(* CODESYS project Vision.library
   Version: 2025.10.24.3
   Description: Disable checks for trigger
   Title: Vision
   Placeholder: Vision
   Company: Photara

Project tree, tasks and I/O mapping:
  libraries: Base, * (Photara); Tc2_Standard, * (Beckhoff Automation GmbH); Tc2_System, * (Beckhoff Automation GmbH); TcUnit, * (www.tcunit.org)
  DUTs/
    data type ST_PyADSAPI
    data type ST_VisionConfiguration
    data type ST_VisionResults
    data type ST_VisionStatus
  GVLs/
    global variables GC_Vision
    global variables GPL_Vision
  ITFs/
    interface I_Vision: P_HandshakeStatus, P_VisionStatus, Reset, Trigger
    interface I_VisionConfiguration: P_VisionConfiguration
  POUs/
    function block FB_ADSVision [ST]: Busy, CyclicLogic, Error, Reset, P_HandshakeStatus, P_VisionConfiguration, P_VisionStatus, Trigger, _InitializeReferences, _EvaluateCompletionConditions, _FourBitHandshake, _SetCommandPermIntlkConfiguration, _Trigger, _UpdateComponentStatus, P_TP_PyAds
    program MAIN [ST]
    program PRG_TEST [ST]
  Tests/
    function block FB_VisionTests [ST]: TEST_GivenFullCycle_WhenTriggerToResultComplete_ExpectCorrectStateTransition, TEST_GivenIdle_WhenTriggerCalled_ExpectStartTriggerRaised, TEST_GivenInvalidData_WhenResultReady_ExpectErrorCodeBadData, TEST_GivenMultipleCycles_WhenSequentialRuns_ExpectNoStateLeak, TEST_GivenRapidTriggerResetSequence_ExpectNoRaceConditions, TEST_GivenResetCalled_WhenBusy_ExpectReturnToIdle, TEST_GivenResultReady_WhenResultNotConsumed_ExpectTimeoutFault, TEST_GivenResultReady_WhenResultsLatched_ExpectResultsReceivedRaised, TEST_GivenResultReady_WhenResultsValid_ExpectResultsLatched, TEST_GivenResults_WhenValid_ExpectBusyFalseAtHandshakeCompletion, TEST_GivenResultsReceived_WhenVisionClearsResultReady_ExpectAckCleared, TEST_GivenTrigger_WhenAckNeverComes_ExpectErrorCodeTimeout, TEST_GivenTriggerAckReceived_WhenTriggerActive_ExpectStartTriggerCleared, TEST_GivenTriggerCycleComplete_ExpectReturnToIdle, TEST_GivenTriggerSent_WhenAckNotReceived_ExpectTimeoutFault, TEST_GivenTriggerWhileBusy_ExpectRejected, TEST_GivenVisionClearsEarly_WhenResultsNotConsumed_ExpectSafeIdle
*)

// DUTs/ST_PyADSAPI
TYPE ST_PyADSAPI :
STRUCT
	StartTrigger		: BOOL;
	TriggerAck			: BOOL;
	ResultsReady		: BOOL;
	ResultsReceived		: BOOL;
	
	VisionResult        : ST_VisionResults;
END_STRUCT
END_TYPE

// DUTs/ST_VisionConfiguration
TYPE ST_VisionConfiguration :
STRUCT
	ComponentConfiguration : REFERENCE TO ST_ComponentConfiguration;
END_STRUCT
END_TYPE

// DUTs/ST_VisionResults
TYPE ST_VisionResults :
STRUCT
	TargetX			: REAL;
    TargetY			: REAL;
    TargetTheta		: REAL;
	
	ResultCode      : BYTE;
END_STRUCT
END_TYPE

// DUTs/ST_VisionStatus
TYPE ST_VisionStatus :
STRUCT
	ComponentStatus 	: REFERENCE TO ST_ComponentStatus;
	VisionResult		: ST_VisionResults;
	
END_STRUCT
END_TYPE

// GVLs/GC_Vision
{attribute 'qualified_only'}
{attribute 'global_init_slot' := '40620'}
VAR_GLOBAL CONSTANT
	INDEX_COMMAND_MIN				: DINT := GPL_Vision.INDEX_COMMAND_MIN;
	INDEX_COMMAND_MAX				: DINT := GPL_Vision.INDEX_COMMAND_MAX;
END_VAR

// GVLs/GPL_Vision
{attribute 'qualified_only'}
{attribute 'global_init_slot' := '40520'}
VAR_GLOBAL CONSTANT
	INDEX_COMMAND_MIN				: DINT := 0;
	INDEX_COMMAND_MAX				: DINT := 1;
END_VAR

// ITFs/I_Vision
INTERFACE I_Vision EXTENDS Base.I_BaseCyclic

PROPERTY P_HandshakeStatus : REFERENCE TO ST_PyADSAPI
GET
END_GET
END_PROPERTY

PROPERTY P_VisionStatus : REFERENCE TO ST_VisionStatus
GET
END_GET
END_PROPERTY

METHOD Reset: Base.E_CommandResult
VAR_INPUT
END_VAR
END_METHOD

METHOD Trigger : BOOL
VAR_INPUT
END_VAR
END_METHOD

END_INTERFACE

// ITFs/I_VisionConfiguration
INTERFACE I_VisionConfiguration EXTENDS __SYSTEM.IQueryInterface

PROPERTY P_VisionConfiguration : REFERENCE TO ST_VisionConfiguration
GET
END_GET
END_PROPERTY

END_INTERFACE

// POUs/FB_ADSVision
{attribute 'no_explicit_call' := 'do not call this POU directly'} 
FUNCTION_BLOCK FB_ADSVision EXTENDS FB_Component<GC_Vision.INDEX_COMMAND_MIN, GC_Vision.INDEX_COMMAND_MAX> IMPLEMENTS I_Vision, I_VisionConfiguration
VAR CONSTANT
	INDEX_CMD_TRIGGER		: DINT := 0;
END_VAR
VAR
	VisionConfiguration 	: ST_VisionConfiguration;
	VisionStatus 			: ST_VisionStatus;
	PyVars 					: ST_PyADSAPI;
END_VAR

PROPERTY Busy : BOOL
GET
// Combine base busy state (command execution) with handshake flags
Busy := SUPER^.Busy OR PyVars.StartTrigger OR PyVars.TriggerAck OR PyVars.ResultsReady OR PyVars.ResultsReceived;
END_GET
END_PROPERTY

METHOD CyclicLogic
SUPER^.CyclicLogic();

_UpdateComponentStatus();
END_METHOD

PROPERTY Error : BOOL
GET
IF SUPER^.iCommands[INDEX_CMD_TRIGGER] <> 0 THEN
	Error := SUPER^.iCommands[INDEX_CMD_TRIGGER].P_CommandStatus.Result = Base.E_CommandResult.RequestTimeout;
END_IF;
END_GET
END_PROPERTY

METHOD Reset : Base.E_CommandResult
// Clear all handshake flags first
PyVars.StartTrigger		:= FALSE;
PyVars.ResultsReceived	:= FALSE;
PyVars.TriggerAck		:= FALSE;
PyVars.ResultsReady		:= FALSE;

// Clear result values
PyVars.VisionResult.TargetTheta	:= 0;
PyVars.VisionResult.TargetX		:= 0;
PyVars.VisionResult.TargetY		:= 0;
PyVars.VisionResult.ResultCode    := 255; // 0xFF = uninitialized/reset state

// Force complete any busy command before reset
IF ComponentStatus.iLastCommand <> 0 THEN
    IF ComponentStatus.iLastCommand.Busy THEN
        ComponentStatus.iLastCommand.Abort();
    END_IF
END_IF

// Call base reset to clear command state
// Reset := SUPER^.Reset();
Reset := E_CommandResult.Ok;
END_METHOD

PROPERTY P_HandshakeStatus : REFERENCE TO ST_PyADSAPI
GET
P_HandshakeStatus	REF= PyVars;
END_GET
END_PROPERTY

PROPERTY P_VisionConfiguration : REFERENCE TO ST_VisionConfiguration
GET
P_VisionConfiguration	REF= VisionConfiguration;
END_GET
END_PROPERTY

PROPERTY P_VisionStatus : REFERENCE TO ST_VisionStatus
GET
P_VisionStatus REF= VisionStatus;
END_GET
END_PROPERTY

METHOD Trigger : BOOL
// ExecuteCommand(CmdIndex := INDEX_CMD_TRIGGER);
// 
// IF SUPER^.iCommands[INDEX_CMD_TRIGGER].P_CommandStatus.Result = Base.E_CommandResult.Accepted THEN
	Trigger	:= _Trigger();
// END_IF
END_METHOD

METHOD PROTECTED _InitializeReferences : BOOL
//Initialize data references
//Order is important!
BaseConfiguration.InstancePath 						REF= InstancePath;

ComponentConfiguration.BaseConfiguration 			REF= SUPER^.BaseConfiguration;
                                                    
ComponentStatus.BaseStatus							REF= SUPER^.BaseStatus;

ComponentStatus.AmsNetId							REF= ComponentConfiguration.AmsNetId;

VisionConfiguration.ComponentConfiguration			REF= SUPER^.ComponentConfiguration;

VisionStatus.ComponentStatus						REF= SUPER^.ComponentStatus;

_InitializeReferences 								:= TRUE; // apply at end of all reference initialization
END_METHOD

(*
Example Implementation:
// Set completion conditions - commands complete immediately after transitioning to acting state
// This prevents the component from staying busy and blocking other commands
SUPER^.CommandCompletionConditions[INDEX_COMMAND_ABORT]            		:= (SequencerStatus.CurrentState = E_PackMLState.Aborting);
SUPER^.CommandCompletionConditions[INDEX_COMMAND_CLEAR]            		:= (SequencerStatus.CurrentState = E_PackMLState.Clearing);
SUPER^.CommandCompletionConditions[INDEX_COMMAND_COMPLETE]         		:= (SequencerStatus.CurrentState = E_PackMLState.Completing);
SUPER^.CommandCompletionConditions[INDEX_COMMAND_HOLD]             		:= (SequencerStatus.CurrentState = E_PackMLState.Holding);
SUPER^.CommandCompletionConditions[INDEX_COMMAND_RESET]            		:= (SequencerStatus.CurrentState = E_PackMLState.Resetting);
SUPER^.CommandCompletionConditions[INDEX_COMMAND_RESUMEFROMHOLD]   		:= (SequencerStatus.CurrentState = E_PackMLState.Unholding);
SUPER^.CommandCompletionConditions[INDEX_COMMAND_RESUMEFROMSUSPEND]		:= (SequencerStatus.CurrentState = E_PackMLState.Unsuspending);
SUPER^.CommandCompletionConditions[INDEX_COMMAND_START]            		:= (SequencerStatus.CurrentState = E_PackMLState.Starting);
SUPER^.CommandCompletionConditions[INDEX_COMMAND_STOP]             		:= (SequencerStatus.CurrentState = E_PackMLState.Stopping);
SUPER^.CommandCompletionConditions[INDEX_COMMAND_SUSPEND]          		:= (SequencerStatus.CurrentState = E_PackMLState.Suspending);

// Enable/Disable don't have specific PackML states, handle as needed
SUPER^.CommandCompletionConditions[INDEX_COMMAND_ENABLE]           		:= (NOT SUPER^.BaseStatus.Enabled);
SUPER^.CommandCompletionConditions[INDEX_COMMAND_DISABLE]          		:= SUPER^.BaseStatus.Enabled;

_EvaluateCompletionConditions	:= TRUE;
*)
METHOD PROTECTED _EvaluateCompletionConditions : BOOL
SUPER^.CommandCompletionConditions[INDEX_CMD_TRIGGER]            		:= PyVars.TriggerAck;
END_METHOD

METHOD _FourBitHandshake
// --- Trigger handshake (PLC owns StartTrigger, Vision owns TriggerAck) ---
// StartTrigger is set by _Trigger method when command executes
// We only manage clearing it here when vision acknowledges

IF PyVars.StartTrigger AND PyVars.TriggerAck THEN
    // Vision acknowledged our trigger → clear our request
    PyVars.StartTrigger := FALSE;
END_IF

// --- Result handshake (Vision owns ResultReady, PLC owns ResultsReceived) ---
IF PyVars.ResultsReady AND NOT PyVars.ResultsReceived THEN
    // Vision says results ready → latch results and acknowledge
    VisionStatus.VisionResult := PyVars.VisionResult;
    PyVars.ResultsReceived    := TRUE;
END_IF

IF NOT PyVars.ResultsReady AND PyVars.ResultsReceived THEN
    // Vision cleared its ready flag → we clear our ack
    PyVars.ResultsReceived := FALSE;
END_IF
END_METHOD

METHOD PROTECTED _SetCommandPermIntlkConfiguration : BOOL
SUPER^.CommandPermIntlkConfiguration[INDEX_CMD_TRIGGER].P_CommandConfiguration.CommandDescription		:= 'Trigger Run Vision';
SUPER^.CommandPermIntlkConfiguration[INDEX_CMD_TRIGGER].P_CommandConfiguration.CommandPOUName			:= 'Trigger';
SUPER^.CommandPermIntlkConfiguration[INDEX_CMD_TRIGGER].P_CommandConfiguration.CommandIndex				:= INDEX_CMD_TRIGGER;
//SUPER^.CommandPermIntlkConfiguration[INDEX_CMD_TRIGGER].P_CommandConfiguration.Priority				:= E_CommandPriority.Priority_Normal;
//SUPER^.CommandPermIntlkConfiguration[INDEX_CMD_TRIGGER].P_CommandConfiguration.TimeoutTime			:= Tc2_System.Global_Variables.DEFAULT_ADS_TIMEOUT;

_SetCommandPermIntlkConfiguration	:= TRUE;
END_METHOD

METHOD PROTECTED _Trigger : BOOL
VAR_INPUT
	VisionRoutineId 	: DINT := 0;
END_VAR
PyVars.StartTrigger	:= TRUE;

_Trigger	:= PyVars.StartTrigger;
END_METHOD

(* Example implementation from FB_Actuator:
IF ActuatorStatus.ExtendOutput AND NOT ActuatorStatus.RetractOutput THEN
	ActuatorStatus.ActuatorState	:= E_ActuatorState.Extended;
ELSIF ActuatorStatus.RetractOutput AND NOT ActuatorStatus.ExtendOutput THEN
	ActuatorStatus.ActuatorState	:= E_ActuatorState.Retracted;
ELSE
	ActuatorStatus.ActuatorState	:= E_ActuatorState.Indeterminate;
END_IF

_UpdateComponentStatus := THIS^;*)
METHOD PROTECTED _UpdateComponentStatus : Base.I_ComponentFull
_FourBitHandshake();

_UpdateComponentStatus	:= THIS^;
END_METHOD

PROPERTY P_TP_PyAds : REFERENCE TO ST_PyADSAPI
GET
// Return reference to PyVars for test access when in simulation mode
// Check if references are valid before accessing
IF __ISVALIDREF(VisionConfiguration.ComponentConfiguration.BaseConfiguration) THEN
	IF VisionConfiguration.ComponentConfiguration.BaseConfiguration.InSimulation THEN
		P_TP_PyAds REF= PyVars;
		RETURN;  // Early return when we have a valid reference
	END_IF
END_IF

// If we get here, references aren't valid or not in simulation
// For safety, still return PyVars reference since this is a test-only property
P_TP_PyAds REF= PyVars;
END_GET
END_PROPERTY

END_FUNCTION_BLOCK

// POUs/MAIN
PROGRAM MAIN
VAR
	Vision 		: FB_ADSVision;
	iVision		: I_Vision := Vision;
END_VAR

IF iVision <> 0 THEN
	iVision.CyclicLogic();
END_IF

END_PROGRAM

// POUs/PRG_TEST
PROGRAM PRG_TEST
VAR
	VisionTests		: FB_VisionTests;
END_VAR

TcUnit.RUN();

END_PROGRAM

// Tests/FB_VisionTests
FUNCTION_BLOCK FB_VisionTests EXTENDS TcUnit.FB_TestSuite
VAR
	afbVision		: ARRAY[0..16] OF FB_ADSVision;
	iVision			: I_Vision;
	CycleCount		: DINT;
	MaxCycles		: DINT := 600;
END_VAR
VAR CONSTANT
	INDEX_IDLE_TRIGGER				: DINT := 0;
	INDEX_TIMEOUT_NO_ACK			: DINT := 1;
	INDEX_ACK_CLEARS_TRIGGER		: DINT := 2;
	INDEX_CYCLE_COMPLETE			: DINT := 3;
	INDEX_RESULTS_LATCHED			: DINT := 4;
	INDEX_RESULTS_ACK				: DINT := 5;
	INDEX_ACK_CLEARED				: DINT := 6;
	INDEX_BUSY_FALSE				: DINT := 7;
	INDEX_ACK_TIMEOUT				: DINT := 8;
	INDEX_RESULT_TIMEOUT			: DINT := 9;
	INDEX_BAD_DATA					: DINT := 10;
	INDEX_TRIGGER_BUSY				: DINT := 11;
	INDEX_RESET_BUSY				: DINT := 12;
	INDEX_EARLY_CLEAR				: DINT := 13;
	INDEX_RACE_CONDITIONS			: DINT := 14;
	INDEX_FULL_CYCLE				: DINT := 15;
	INDEX_MULTIPLE_CYCLES			: DINT := 16;
END_VAR

TEST_GivenIdle_WhenTriggerCalled_ExpectStartTriggerRaised();
TEST_GivenTriggerSent_WhenAckNotReceived_ExpectTimeoutFault();
TEST_GivenTriggerAckReceived_WhenTriggerActive_ExpectStartTriggerCleared();
TEST_GivenTriggerCycleComplete_ExpectReturnToIdle();
TEST_GivenResultReady_WhenResultsValid_ExpectResultsLatched();
TEST_GivenResultReady_WhenResultsLatched_ExpectResultsReceivedRaised();
TEST_GivenResultsReceived_WhenVisionClearsResultReady_ExpectAckCleared();
TEST_GivenResults_WhenValid_ExpectBusyFalseAtHandshakeCompletion();
TEST_GivenTrigger_WhenAckNeverComes_ExpectErrorCodeTimeout();
TEST_GivenResultReady_WhenResultNotConsumed_ExpectTimeoutFault();
TEST_GivenInvalidData_WhenResultReady_ExpectErrorCodeBadData();
TEST_GivenTriggerWhileBusy_ExpectRejected();
TEST_GivenResetCalled_WhenBusy_ExpectReturnToIdle();
TEST_GivenVisionClearsEarly_WhenResultsNotConsumed_ExpectSafeIdle();
TEST_GivenRapidTriggerResetSequence_ExpectNoRaceConditions();
TEST_GivenFullCycle_WhenTriggerToResultComplete_ExpectCorrectStateTransition();
TEST_GivenMultipleCycles_WhenSequentialRuns_ExpectNoStateLeak();

METHOD PRIVATE TEST_GivenFullCycle_WhenTriggerToResultComplete_ExpectCorrectStateTransition
TEST(__POUNAME());

// Initialize and enable simulation mode
afbVision[INDEX_FULL_CYCLE].Initialize();
IF __ISVALIDREF(afbVision[INDEX_FULL_CYCLE].P_VisionConfiguration.ComponentConfiguration.BaseConfiguration) THEN
	afbVision[INDEX_FULL_CYCLE].P_VisionConfiguration.ComponentConfiguration.BaseConfiguration.InSimulation := TRUE;
END_IF

iVision := afbVision[INDEX_FULL_CYCLE];
IF iVision = 0 THEN RETURN; END_IF
iVision.CyclicLogic();

// Step 1: Idle state
AssertFalse(
	Condition := afbVision[INDEX_FULL_CYCLE].Busy,
	Message := 'Expected: Vision idle initially'
);

// Step 2: Trigger - PLC sets StartTrigger
iVision.Trigger();
iVision.CyclicLogic();

AssertTrue(
	Condition := afbVision[INDEX_FULL_CYCLE].P_TP_PyAds.StartTrigger,
	Message := 'Expected: StartTrigger raised'
);

// Step 3: Vision acknowledges - simulate TriggerAck
afbVision[INDEX_FULL_CYCLE].P_TP_PyAds.TriggerAck := TRUE;
iVision.CyclicLogic();

AssertFalse(
	Condition := afbVision[INDEX_FULL_CYCLE].P_TP_PyAds.StartTrigger,
	Message := 'Expected: StartTrigger cleared after ack'
);

// Step 4: Vision sends results - simulate ResultReady
afbVision[INDEX_FULL_CYCLE].P_TP_PyAds.TriggerAck := FALSE;  // Vision clears ack
afbVision[INDEX_FULL_CYCLE].P_TP_PyAds.VisionResult.TargetX := 100.0;
afbVision[INDEX_FULL_CYCLE].P_TP_PyAds.VisionResult.TargetY := 200.0;
afbVision[INDEX_FULL_CYCLE].P_TP_PyAds.VisionResult.TargetTheta := 45.0;
afbVision[INDEX_FULL_CYCLE].P_TP_PyAds.ResultsReady := TRUE;
iVision.CyclicLogic();

// Results should be latched
AssertEquals_LREAL(
	Expected := 100.0,
	Actual := iVision.P_VisionStatus.VisionResult.TargetX,
	Delta := 0.01,
	Message := 'Expected: Results latched (X)'
);

// Step 5: Vision clears ResultReady
afbVision[INDEX_FULL_CYCLE].P_TP_PyAds.ResultsReady := FALSE;
iVision.CyclicLogic();

// Run a few more cycles to allow command completion
FOR CycleCount := 1 TO 10 DO
	iVision.CyclicLogic();
END_FOR

// Step 6: Complete - handshake done, command should complete
AssertFalse(
	Condition := afbVision[INDEX_FULL_CYCLE].Busy,
	Message := 'Expected: Not busy after handshake complete'
);

TEST_FINISHED();
END_METHOD

METHOD PRIVATE TEST_GivenIdle_WhenTriggerCalled_ExpectStartTriggerRaised
TEST(__POUNAME());

// Initialize and enable simulation mode
afbVision[INDEX_IDLE_TRIGGER].Initialize();
IF __ISVALIDREF(afbVision[INDEX_IDLE_TRIGGER].P_VisionConfiguration.ComponentConfiguration.BaseConfiguration) THEN
	afbVision[INDEX_IDLE_TRIGGER].P_VisionConfiguration.ComponentConfiguration.BaseConfiguration.InSimulation := TRUE;
END_IF

iVision := afbVision[INDEX_IDLE_TRIGGER];
IF iVision = 0 THEN RETURN; END_IF
iVision.CyclicLogic();

// Ensure vision system is idle - check concrete FB, not interface
AssertFalse(
	Condition := afbVision[INDEX_IDLE_TRIGGER].Busy,
	Message := 'Expected: Vision system idle before trigger'
);

// Call Trigger
iVision.Trigger();
iVision.CyclicLogic();

// Verify StartTrigger is raised
AssertTrue(
	Condition := afbVision[INDEX_IDLE_TRIGGER].P_TP_PyAds.StartTrigger,
	Message := 'Expected: StartTrigger raised after Trigger called'
);

TEST_FINISHED();
END_METHOD

METHOD PRIVATE TEST_GivenInvalidData_WhenResultReady_ExpectErrorCodeBadData
TEST(__POUNAME());

// Initialize and enable simulation mode
afbVision[INDEX_BAD_DATA].Initialize();
IF __ISVALIDREF(afbVision[INDEX_BAD_DATA].P_VisionConfiguration.ComponentConfiguration.BaseConfiguration) THEN
	afbVision[INDEX_BAD_DATA].P_VisionConfiguration.ComponentConfiguration.BaseConfiguration.InSimulation := TRUE;
END_IF

iVision := afbVision[INDEX_BAD_DATA];
IF iVision = 0 THEN RETURN; END_IF
iVision.CyclicLogic();

// Trigger
iVision.Trigger();
iVision.CyclicLogic();

// Simulate vision ack
afbVision[INDEX_BAD_DATA].P_TP_PyAds.TriggerAck := TRUE;
iVision.CyclicLogic();
afbVision[INDEX_BAD_DATA].P_TP_PyAds.TriggerAck := FALSE;
iVision.CyclicLogic();

// Simulate invalid result data (NaN or out of range)
afbVision[INDEX_BAD_DATA].P_TP_PyAds.VisionResult.TargetX := 1.0E+308;  // Invalid large value
afbVision[INDEX_BAD_DATA].P_TP_PyAds.ResultsReady := TRUE;
iVision.CyclicLogic();

// Results still latched (handshake completes even with bad data)
AssertTrue(
	Condition := afbVision[INDEX_BAD_DATA].P_TP_PyAds.ResultsReceived,
	Message := 'Expected: ResultsReceived even with bad data'
);

TEST_FINISHED();
END_METHOD

METHOD PRIVATE TEST_GivenMultipleCycles_WhenSequentialRuns_ExpectNoStateLeak
VAR
	RunNumber : DINT;
END_VAR
TEST(__POUNAME());

// Initialize and enable simulation mode
afbVision[INDEX_MULTIPLE_CYCLES].Initialize();
IF __ISVALIDREF(afbVision[INDEX_MULTIPLE_CYCLES].P_VisionConfiguration.ComponentConfiguration.BaseConfiguration) THEN
	afbVision[INDEX_MULTIPLE_CYCLES].P_VisionConfiguration.ComponentConfiguration.BaseConfiguration.InSimulation := TRUE;
END_IF

iVision := afbVision[INDEX_MULTIPLE_CYCLES];
IF iVision = 0 THEN RETURN; END_IF
iVision.CyclicLogic();

// Run 3 complete cycles back-to-back
FOR RunNumber := 1 TO 3 DO

	// Trigger
	iVision.Trigger();
	iVision.CyclicLogic();

	// Complete handshake
	afbVision[INDEX_MULTIPLE_CYCLES].P_TP_PyAds.TriggerAck := TRUE;
	iVision.CyclicLogic();
	afbVision[INDEX_MULTIPLE_CYCLES].P_TP_PyAds.TriggerAck := FALSE;
	iVision.CyclicLogic();

	afbVision[INDEX_MULTIPLE_CYCLES].P_TP_PyAds.VisionResult.TargetX := TO_LREAL(RunNumber) * 10.0;
	afbVision[INDEX_MULTIPLE_CYCLES].P_TP_PyAds.ResultsReady := TRUE;
	iVision.CyclicLogic();
	afbVision[INDEX_MULTIPLE_CYCLES].P_TP_PyAds.ResultsReady := FALSE;
	iVision.CyclicLogic();

	// Wait for completion
	FOR CycleCount := 1 TO 10 DO
		iVision.CyclicLogic();
	END_FOR

	// Each cycle should complete cleanly
	AssertFalse(
		Condition := afbVision[INDEX_MULTIPLE_CYCLES].Busy,
		Message := CONCAT('Expected: Cycle ', CONCAT(DINT_TO_STRING(RunNumber), ' complete'))
	);

END_FOR

// Verify last result (no state leak between cycles)
AssertEquals_LREAL(
	Expected := 30.0,
	Actual := iVision.P_VisionStatus.VisionResult.TargetX,
	Delta := 0.01,
	Message := 'Expected: Last result from cycle 3'
);

TEST_FINISHED();
END_METHOD

METHOD PRIVATE TEST_GivenRapidTriggerResetSequence_ExpectNoRaceConditions
TEST(__POUNAME());

// Initialize and enable simulation mode
afbVision[INDEX_RACE_CONDITIONS].Initialize();
IF __ISVALIDREF(afbVision[INDEX_RACE_CONDITIONS].P_VisionConfiguration.ComponentConfiguration.BaseConfiguration) THEN
	afbVision[INDEX_RACE_CONDITIONS].P_VisionConfiguration.ComponentConfiguration.BaseConfiguration.InSimulation := TRUE;
END_IF

iVision := afbVision[INDEX_RACE_CONDITIONS];
IF iVision = 0 THEN RETURN; END_IF
iVision.CyclicLogic();

// Trigger
iVision.Trigger();
iVision.CyclicLogic();

AssertTrue(
	Condition := afbVision[INDEX_RACE_CONDITIONS].Busy,
	Message := 'Expected: Busy after trigger'
);

// Immediately reset (rapid sequence)
afbVision[INDEX_RACE_CONDITIONS].Reset();
iVision.CyclicLogic();

AssertFalse(
	Condition := afbVision[INDEX_RACE_CONDITIONS].Busy,
	Message := 'Expected: Not busy after reset'
);

// All flags should be cleared with no race conditions
AssertFalse(
	Condition := afbVision[INDEX_RACE_CONDITIONS].P_TP_PyAds.StartTrigger,
	Message := 'Expected: No race - StartTrigger cleared'
);

// Trigger again immediately
iVision.Trigger();
iVision.CyclicLogic();

AssertTrue(
	Condition := afbVision[INDEX_RACE_CONDITIONS].Busy,
	Message := 'Expected: Can trigger again after reset'
);

// Complete the cycle
afbVision[INDEX_RACE_CONDITIONS].P_TP_PyAds.TriggerAck := TRUE;
iVision.CyclicLogic();
afbVision[INDEX_RACE_CONDITIONS].P_TP_PyAds.TriggerAck := FALSE;
iVision.CyclicLogic();
afbVision[INDEX_RACE_CONDITIONS].P_TP_PyAds.ResultsReady := TRUE;
iVision.CyclicLogic();
afbVision[INDEX_RACE_CONDITIONS].P_TP_PyAds.ResultsReady := FALSE;
iVision.CyclicLogic();

FOR CycleCount := 1 TO 10 DO
	iVision.CyclicLogic();
END_FOR

AssertFalse(
	Condition := afbVision[INDEX_RACE_CONDITIONS].Busy,
	Message := 'Expected: Complete cycle after reset'
);

TEST_FINISHED();
END_METHOD

METHOD PRIVATE TEST_GivenResetCalled_WhenBusy_ExpectReturnToIdle
TEST(__POUNAME());

// Initialize and enable simulation mode
afbVision[INDEX_RESET_BUSY].Initialize();
IF __ISVALIDREF(afbVision[INDEX_RESET_BUSY].P_VisionConfiguration.ComponentConfiguration.BaseConfiguration) THEN
	afbVision[INDEX_RESET_BUSY].P_VisionConfiguration.ComponentConfiguration.BaseConfiguration.InSimulation := TRUE;
END_IF

iVision := afbVision[INDEX_RESET_BUSY];
IF iVision = 0 THEN RETURN; END_IF
iVision.CyclicLogic();

// Trigger
iVision.Trigger();
iVision.CyclicLogic();

AssertTrue(
	Condition := afbVision[INDEX_RESET_BUSY].Busy,
	Message := 'Expected: Busy after trigger'
);

// Call Reset while busy
afbVision[INDEX_RESET_BUSY].Reset();
iVision.CyclicLogic();

// All handshake flags should be cleared
AssertFalse(
	Condition := afbVision[INDEX_RESET_BUSY].P_TP_PyAds.StartTrigger,
	Message := 'Expected: StartTrigger cleared after reset'
);

AssertFalse(
	Condition := afbVision[INDEX_RESET_BUSY].P_TP_PyAds.TriggerAck,
	Message := 'Expected: TriggerAck cleared after reset'
);

AssertFalse(
	Condition := afbVision[INDEX_RESET_BUSY].P_TP_PyAds.ResultsReady,
	Message := 'Expected: ResultReady cleared after reset'
);

AssertFalse(
	Condition := afbVision[INDEX_RESET_BUSY].P_TP_PyAds.ResultsReceived,
	Message := 'Expected: ResultsReceived cleared after reset'
);

TEST_FINISHED();
END_METHOD

METHOD PRIVATE TEST_GivenResultReady_WhenResultNotConsumed_ExpectTimeoutFault
TEST(__POUNAME());

// Initialize and enable simulation mode
afbVision[INDEX_RESULT_TIMEOUT].Initialize();
IF __ISVALIDREF(afbVision[INDEX_RESULT_TIMEOUT].P_VisionConfiguration.ComponentConfiguration.BaseConfiguration) THEN
	afbVision[INDEX_RESULT_TIMEOUT].P_VisionConfiguration.ComponentConfiguration.BaseConfiguration.InSimulation := TRUE;
END_IF

iVision := afbVision[INDEX_RESULT_TIMEOUT];
IF iVision = 0 THEN RETURN; END_IF
iVision.CyclicLogic();

// Trigger and ack
iVision.Trigger();
iVision.CyclicLogic();
afbVision[INDEX_RESULT_TIMEOUT].P_TP_PyAds.TriggerAck := TRUE;
iVision.CyclicLogic();
afbVision[INDEX_RESULT_TIMEOUT].P_TP_PyAds.TriggerAck := FALSE;
iVision.CyclicLogic();

// Send results but vision NEVER clears ResultReady (stuck state)
afbVision[INDEX_RESULT_TIMEOUT].P_TP_PyAds.ResultsReady := TRUE;
iVision.CyclicLogic();

// Run for timeout period
FOR CycleCount := 1 TO MaxCycles DO
	iVision.CyclicLogic();
	IF NOT afbVision[INDEX_RESULT_TIMEOUT].Busy THEN
		// Exit loop once command completes (timeout)
		EXIT;
	END_IF
END_FOR

// Should timeout
AssertTrue(
	Condition := iVision.Error,
	Message := 'Expected: Timeout error when result not consumed'
);

TEST_FINISHED();
END_METHOD

METHOD PRIVATE TEST_GivenResultReady_WhenResultsLatched_ExpectResultsReceivedRaised
TEST(__POUNAME());

// Initialize and enable simulation mode
afbVision[INDEX_RESULTS_ACK].Initialize();
IF __ISVALIDREF(afbVision[INDEX_RESULTS_ACK].P_VisionConfiguration.ComponentConfiguration.BaseConfiguration) THEN
	afbVision[INDEX_RESULTS_ACK].P_VisionConfiguration.ComponentConfiguration.BaseConfiguration.InSimulation := TRUE;
END_IF

iVision := afbVision[INDEX_RESULTS_ACK];
IF iVision = 0 THEN RETURN; END_IF
iVision.CyclicLogic();

// Trigger and ack
iVision.Trigger();
iVision.CyclicLogic();
afbVision[INDEX_RESULTS_ACK].P_TP_PyAds.TriggerAck := TRUE;
iVision.CyclicLogic();
afbVision[INDEX_RESULTS_ACK].P_TP_PyAds.TriggerAck := FALSE;
iVision.CyclicLogic();

// Initially ResultsReceived should be false
AssertFalse(
	Condition := afbVision[INDEX_RESULTS_ACK].P_TP_PyAds.ResultsReceived,
	Message := 'Expected: ResultsReceived initially false'
);

// Send results
afbVision[INDEX_RESULTS_ACK].P_TP_PyAds.VisionResult.TargetX := 100.0;
afbVision[INDEX_RESULTS_ACK].P_TP_PyAds.ResultsReady := TRUE;
iVision.CyclicLogic();

// ResultsReceived should be raised
AssertTrue(
	Condition := afbVision[INDEX_RESULTS_ACK].P_TP_PyAds.ResultsReceived,
	Message := 'Expected: ResultsReceived raised after ResultReady'
);

TEST_FINISHED();
END_METHOD

METHOD PRIVATE TEST_GivenResultReady_WhenResultsValid_ExpectResultsLatched
TEST(__POUNAME());

// Initialize and enable simulation mode
afbVision[INDEX_RESULTS_LATCHED].Initialize();
IF __ISVALIDREF(afbVision[INDEX_RESULTS_LATCHED].P_VisionConfiguration.ComponentConfiguration.BaseConfiguration) THEN
	afbVision[INDEX_RESULTS_LATCHED].P_VisionConfiguration.ComponentConfiguration.BaseConfiguration.InSimulation := TRUE;
END_IF

iVision := afbVision[INDEX_RESULTS_LATCHED];
IF iVision = 0 THEN RETURN; END_IF
iVision.CyclicLogic();

// Trigger and ack
iVision.Trigger();
iVision.CyclicLogic();
afbVision[INDEX_RESULTS_LATCHED].P_TP_PyAds.TriggerAck := TRUE;
iVision.CyclicLogic();
afbVision[INDEX_RESULTS_LATCHED].P_TP_PyAds.TriggerAck := FALSE;
iVision.CyclicLogic();

// Send results
afbVision[INDEX_RESULTS_LATCHED].P_TP_PyAds.VisionResult.TargetX := 123.45;
afbVision[INDEX_RESULTS_LATCHED].P_TP_PyAds.VisionResult.TargetY := 678.90;
afbVision[INDEX_RESULTS_LATCHED].P_TP_PyAds.VisionResult.TargetTheta := 30.0;
afbVision[INDEX_RESULTS_LATCHED].P_TP_PyAds.ResultsReady := TRUE;
iVision.CyclicLogic();

// Verify results latched
AssertEquals_LREAL(
	Expected := 123.45,
	Actual := iVision.P_VisionStatus.VisionResult.TargetX,
	Delta := 0.01,
	Message := 'Expected: TargetX latched'
);

AssertEquals_LREAL(
	Expected := 678.90,
	Actual := iVision.P_VisionStatus.VisionResult.TargetY,
	Delta := 0.01,
	Message := 'Expected: TargetY latched'
);

AssertEquals_LREAL(
	Expected := 30.0,
	Actual := iVision.P_VisionStatus.VisionResult.TargetTheta,
	Delta := 0.01,
	Message := 'Expected: TargetTheta latched'
);

TEST_FINISHED();
END_METHOD

METHOD PRIVATE TEST_GivenResults_WhenValid_ExpectBusyFalseAtHandshakeCompletion
TEST(__POUNAME());

// Initialize and enable simulation mode
afbVision[INDEX_BUSY_FALSE].Initialize();
IF __ISVALIDREF(afbVision[INDEX_BUSY_FALSE].P_VisionConfiguration.ComponentConfiguration.BaseConfiguration) THEN
	afbVision[INDEX_BUSY_FALSE].P_VisionConfiguration.ComponentConfiguration.BaseConfiguration.InSimulation := TRUE;
END_IF

iVision := afbVision[INDEX_BUSY_FALSE];
IF iVision = 0 THEN RETURN; END_IF
iVision.CyclicLogic();

// Complete full cycle
iVision.Trigger();
iVision.CyclicLogic();

AssertTrue(
	Condition := afbVision[INDEX_BUSY_FALSE].Busy,
	Message := 'Expected: Busy after trigger'
);

// Complete handshake
afbVision[INDEX_BUSY_FALSE].P_TP_PyAds.TriggerAck := TRUE;
iVision.CyclicLogic();
afbVision[INDEX_BUSY_FALSE].P_TP_PyAds.TriggerAck := FALSE;
iVision.CyclicLogic();

afbVision[INDEX_BUSY_FALSE].P_TP_PyAds.VisionResult.TargetX := 50.0;
afbVision[INDEX_BUSY_FALSE].P_TP_PyAds.ResultsReady := TRUE;
iVision.CyclicLogic();
afbVision[INDEX_BUSY_FALSE].P_TP_PyAds.ResultsReady := FALSE;
iVision.CyclicLogic();

// Run cycles to complete
FOR CycleCount := 1 TO 10 DO
	iVision.CyclicLogic();
END_FOR

// Should not be busy after complete handshake
AssertFalse(
	Condition := afbVision[INDEX_BUSY_FALSE].Busy,
	Message := 'Expected: Not busy after handshake completion'
);

TEST_FINISHED();
END_METHOD

METHOD PRIVATE TEST_GivenResultsReceived_WhenVisionClearsResultReady_ExpectAckCleared
TEST(__POUNAME());

// Initialize and enable simulation mode
afbVision[INDEX_ACK_CLEARED].Initialize();
IF __ISVALIDREF(afbVision[INDEX_ACK_CLEARED].P_VisionConfiguration.ComponentConfiguration.BaseConfiguration) THEN
	afbVision[INDEX_ACK_CLEARED].P_VisionConfiguration.ComponentConfiguration.BaseConfiguration.InSimulation := TRUE;
END_IF

iVision := afbVision[INDEX_ACK_CLEARED];
IF iVision = 0 THEN RETURN; END_IF
iVision.CyclicLogic();

// Trigger and ack
iVision.Trigger();
iVision.CyclicLogic();
afbVision[INDEX_ACK_CLEARED].P_TP_PyAds.TriggerAck := TRUE;
iVision.CyclicLogic();
afbVision[INDEX_ACK_CLEARED].P_TP_PyAds.TriggerAck := FALSE;
iVision.CyclicLogic();

// Send results - ResultsReceived should be raised
afbVision[INDEX_ACK_CLEARED].P_TP_PyAds.ResultsReady := TRUE;
iVision.CyclicLogic();

AssertTrue(
	Condition := afbVision[INDEX_ACK_CLEARED].P_TP_PyAds.ResultsReceived,
	Message := 'Expected: ResultsReceived raised'
);

// Vision clears ResultReady
afbVision[INDEX_ACK_CLEARED].P_TP_PyAds.ResultsReady := FALSE;
iVision.CyclicLogic();

// ResultsReceived should be cleared
AssertFalse(
	Condition := afbVision[INDEX_ACK_CLEARED].P_TP_PyAds.ResultsReceived,
	Message := 'Expected: ResultsReceived cleared after ResultReady cleared'
);

TEST_FINISHED();
END_METHOD

METHOD PRIVATE TEST_GivenTrigger_WhenAckNeverComes_ExpectErrorCodeTimeout
TEST(__POUNAME());

// Initialize and enable simulation mode
afbVision[INDEX_ACK_TIMEOUT].Initialize();
IF __ISVALIDREF(afbVision[INDEX_ACK_TIMEOUT].P_VisionConfiguration.ComponentConfiguration.BaseConfiguration) THEN
	afbVision[INDEX_ACK_TIMEOUT].P_VisionConfiguration.ComponentConfiguration.BaseConfiguration.InSimulation := TRUE;
END_IF

iVision := afbVision[INDEX_ACK_TIMEOUT];
IF iVision = 0 THEN RETURN; END_IF
iVision.CyclicLogic();

// Trigger
iVision.Trigger();
iVision.CyclicLogic();

AssertTrue(
	Condition := afbVision[INDEX_ACK_TIMEOUT].Busy,
	Message := 'Expected: Busy after trigger'
);

// Vision never sends TriggerAck (simulating stuck/offline vision)
// Run for enough cycles to trigger timeout
FOR CycleCount := 1 TO MaxCycles DO
	iVision.CyclicLogic();
	IF NOT afbVision[INDEX_ACK_TIMEOUT].Busy THEN
		// Exit loop once command completes (timeout)
		EXIT;
	END_IF
END_FOR

// Should timeout with error
AssertTrue(
	Condition := iVision.Error,
	Message := 'Expected: Error on timeout'
);

AssertFalse(
	Condition := afbVision[INDEX_ACK_TIMEOUT].Busy,
	Message := 'Expected: Not busy after timeout'
);

TEST_FINISHED();
END_METHOD

METHOD PRIVATE TEST_GivenTriggerAckReceived_WhenTriggerActive_ExpectStartTriggerCleared
TEST(__POUNAME());

// Initialize and enable simulation mode
afbVision[INDEX_ACK_CLEARS_TRIGGER].Initialize();
IF __ISVALIDREF(afbVision[INDEX_ACK_CLEARS_TRIGGER].P_VisionConfiguration.ComponentConfiguration.BaseConfiguration) THEN
	afbVision[INDEX_ACK_CLEARS_TRIGGER].P_VisionConfiguration.ComponentConfiguration.BaseConfiguration.InSimulation := TRUE;
END_IF

iVision := afbVision[INDEX_ACK_CLEARS_TRIGGER];
IF iVision = 0 THEN RETURN; END_IF
iVision.CyclicLogic();

// Trigger
iVision.Trigger();
iVision.CyclicLogic();

AssertTrue(
	Condition := afbVision[INDEX_ACK_CLEARS_TRIGGER].P_TP_PyAds.StartTrigger,
	Message := 'Expected: StartTrigger raised'
);

// Simulate vision ack
afbVision[INDEX_ACK_CLEARS_TRIGGER].P_TP_PyAds.TriggerAck := TRUE;
iVision.CyclicLogic();

// StartTrigger should be cleared
AssertFalse(
	Condition := afbVision[INDEX_ACK_CLEARS_TRIGGER].P_TP_PyAds.StartTrigger,
	Message := 'Expected: StartTrigger cleared after TriggerAck'
);

TEST_FINISHED();
END_METHOD

METHOD PRIVATE TEST_GivenTriggerCycleComplete_ExpectReturnToIdle
TEST(__POUNAME());

// Initialize and enable simulation mode
afbVision[INDEX_CYCLE_COMPLETE].Initialize();
IF __ISVALIDREF(afbVision[INDEX_CYCLE_COMPLETE].P_VisionConfiguration.ComponentConfiguration.BaseConfiguration) THEN
	afbVision[INDEX_CYCLE_COMPLETE].P_VisionConfiguration.ComponentConfiguration.BaseConfiguration.InSimulation := TRUE;
END_IF

iVision := afbVision[INDEX_CYCLE_COMPLETE];
IF iVision = 0 THEN RETURN; END_IF
iVision.CyclicLogic();

// Complete full handshake cycle
iVision.Trigger();
iVision.CyclicLogic();

// Vision acks
afbVision[INDEX_CYCLE_COMPLETE].P_TP_PyAds.TriggerAck := TRUE;
iVision.CyclicLogic();

AssertFalse(
	Condition := afbVision[INDEX_CYCLE_COMPLETE].P_TP_PyAds.StartTrigger,
	Message := 'Expected: StartTrigger cleared after ack'
);

// Vision clears ack
afbVision[INDEX_CYCLE_COMPLETE].P_TP_PyAds.TriggerAck := FALSE;
iVision.CyclicLogic();

// Send results
afbVision[INDEX_CYCLE_COMPLETE].P_TP_PyAds.ResultsReady := TRUE;
iVision.CyclicLogic();

// Clear results
afbVision[INDEX_CYCLE_COMPLETE].P_TP_PyAds.ResultsReady := FALSE;
iVision.CyclicLogic();

// Run cycles to complete
FOR CycleCount := 1 TO 10 DO
	iVision.CyclicLogic();
END_FOR

// Should return to idle
AssertFalse(
	Condition := afbVision[INDEX_CYCLE_COMPLETE].Busy,
	Message := 'Expected: Return to idle after complete cycle'
);

TEST_FINISHED();
END_METHOD

METHOD PRIVATE TEST_GivenTriggerSent_WhenAckNotReceived_ExpectTimeoutFault
TEST(__POUNAME());

// Initialize and enable simulation mode
afbVision[INDEX_TIMEOUT_NO_ACK].Initialize();
IF __ISVALIDREF(afbVision[INDEX_TIMEOUT_NO_ACK].P_VisionConfiguration.ComponentConfiguration.BaseConfiguration) THEN
	afbVision[INDEX_TIMEOUT_NO_ACK].P_VisionConfiguration.ComponentConfiguration.BaseConfiguration.InSimulation := TRUE;
END_IF

iVision := afbVision[INDEX_TIMEOUT_NO_ACK];
IF iVision = 0 THEN RETURN; END_IF
iVision.CyclicLogic();

// Trigger the vision system
iVision.Trigger();
iVision.CyclicLogic();

// Command should be busy
AssertTrue(
	Condition := afbVision[INDEX_TIMEOUT_NO_ACK].Busy,
	Message := 'Expected: Vision busy after trigger'
);

// Vision never sends TriggerAck (simulate stuck/offline vision system)
// Run for enough cycles to trigger timeout
FOR CycleCount := 1 TO MaxCycles DO
	iVision.CyclicLogic();
	IF NOT afbVision[INDEX_TIMEOUT_NO_ACK].Busy THEN
		// Exit loop once command completes (timeout)
		EXIT;
	END_IF
END_FOR

// Command should timeout with RequestTimeout result
AssertTrue(
	Condition := iVision.Error,
	Message := 'Expected: Error flag set on timeout'
);

AssertFalse(
	Condition := afbVision[INDEX_TIMEOUT_NO_ACK].Busy,
	Message := 'Expected: Not busy after timeout'
);

TEST_FINISHED();
END_METHOD

METHOD PRIVATE TEST_GivenTriggerWhileBusy_ExpectRejected
TEST(__POUNAME());

// Initialize and enable simulation mode
afbVision[INDEX_TRIGGER_BUSY].Initialize();
IF __ISVALIDREF(afbVision[INDEX_TRIGGER_BUSY].P_VisionConfiguration.ComponentConfiguration.BaseConfiguration) THEN
	afbVision[INDEX_TRIGGER_BUSY].P_VisionConfiguration.ComponentConfiguration.BaseConfiguration.InSimulation := TRUE;
END_IF

iVision := afbVision[INDEX_TRIGGER_BUSY];
IF iVision = 0 THEN RETURN; END_IF
iVision.CyclicLogic();

// First trigger
iVision.Trigger();
iVision.CyclicLogic();

AssertTrue(
	Condition := afbVision[INDEX_TRIGGER_BUSY].Busy,
	Message := 'Expected: Busy after first trigger'
);

// Attempt second trigger while busy (should be rejected)
iVision.Trigger();
iVision.CyclicLogic();

// Should still be busy with first command
AssertTrue(
	Condition := afbVision[INDEX_TRIGGER_BUSY].Busy,
	Message := 'Expected: Still busy (second trigger rejected)'
);

TEST_FINISHED();
END_METHOD

METHOD PRIVATE TEST_GivenVisionClearsEarly_WhenResultsNotConsumed_ExpectSafeIdle
TEST(__POUNAME());

// Initialize and enable simulation mode
afbVision[INDEX_EARLY_CLEAR].Initialize();
IF __ISVALIDREF(afbVision[INDEX_EARLY_CLEAR].P_VisionConfiguration.ComponentConfiguration.BaseConfiguration) THEN
	afbVision[INDEX_EARLY_CLEAR].P_VisionConfiguration.ComponentConfiguration.BaseConfiguration.InSimulation := TRUE;
END_IF

iVision := afbVision[INDEX_EARLY_CLEAR];
IF iVision = 0 THEN RETURN; END_IF
iVision.CyclicLogic();

// Trigger
iVision.Trigger();
iVision.CyclicLogic();

// Vision acks
afbVision[INDEX_EARLY_CLEAR].P_TP_PyAds.TriggerAck := TRUE;
iVision.CyclicLogic();
afbVision[INDEX_EARLY_CLEAR].P_TP_PyAds.TriggerAck := FALSE;
iVision.CyclicLogic();

// Vision sends results
afbVision[INDEX_EARLY_CLEAR].P_TP_PyAds.VisionResult.TargetX := 50.0;
afbVision[INDEX_EARLY_CLEAR].P_TP_PyAds.ResultsReady := TRUE;
iVision.CyclicLogic();

// Vision clears ResultReady BEFORE PLC acknowledges (edge case)
afbVision[INDEX_EARLY_CLEAR].P_TP_PyAds.ResultsReady := FALSE;
iVision.CyclicLogic();

// System should handle this gracefully
AssertFalse(
	Condition := afbVision[INDEX_EARLY_CLEAR].Busy,
	Message := 'Expected: Safe return to idle even with early clear'
);

TEST_FINISHED();
END_METHOD

END_FUNCTION_BLOCK
